{attribute addProperty BoxType "EP2328-1061-0016"}
{attribute addProperty Id "DI_X01_Pin4_InputAT %I*DI_X01_Pin4_Input_E4AEF59E810DI_X01_Pin2_InputAT %I*DI_X01_Pin2_Input_E4AEF59E810DI_X02_Pin4_InputAT %I*DI_X02_Pin4_Input_E4AEF59E810DI_X02_Pin2_InputAT %I*DI_X02_Pin2_Input_E4AEF59E810DO_X03_Pin4_OutputAT %Q*DO_X03_Pin4_Output_7F374EB0810DO_X03_Pin2_OutputAT %Q*DO_X03_Pin2_Output_7F374EB0810DO_X04_Pin4_OutputAT %Q*DO_X04_Pin4_Output_7F374EB0810DO_X04_Pin2_OutputAT %Q*DO_X04_Pin2_Output_7F374EB0810WcStateAT %I*WcState_F855686C1620InfoDataAT %I*InfoData_192954DE1620"}
{attribute addProperty CRC "3768556029"}
{attribute addProperty SizeInBites "96"}
{attribute addProperty SizeInBytes "12"}
TYPE EP2328_6092ACCC :
STRUCT
	{attribute addProperty Name "DI_X01_Pin4_Input"}
	DI_X01_Pin4_Input : DI_X01_Pin4_Input_E4AEF59E;
	{attribute addProperty Name "DI_X01_Pin2_Input"}
	DI_X01_Pin2_Input : DI_X01_Pin2_Input_E4AEF59E;
	{attribute addProperty Name "DI_X02_Pin4_Input"}
	DI_X02_Pin4_Input : DI_X02_Pin4_Input_E4AEF59E;
	{attribute addProperty Name "DI_X02_Pin2_Input"}
	DI_X02_Pin2_Input : DI_X02_Pin2_Input_E4AEF59E;
	{attribute addProperty Name "DO_X03_Pin4_Output"}
	DO_X03_Pin4_Output : DO_X03_Pin4_Output_7F374EB0;
	{attribute addProperty Name "DO_X03_Pin2_Output"}
	DO_X03_Pin2_Output : DO_X03_Pin2_Output_7F374EB0;
	{attribute addProperty Name "DO_X04_Pin4_Output"}
	DO_X04_Pin4_Output : DO_X04_Pin4_Output_7F374EB0;
	{attribute addProperty Name "DO_X04_Pin2_Output"}
	DO_X04_Pin2_Output : DO_X04_Pin2_Output_7F374EB0;
	{attribute addProperty Name "WcState"}
	WcState : WcState_F855686C;
	{attribute addProperty Name "InfoData"}
	InfoData : InfoData_192954DE;
END_STRUCT
END_TYPE

(* stored: Version 1.2.0.0, ProductVersion 3.1.4024.9
   DUT EP2328_6092ACCC: Id {4048953e-6aca-4a97-b35e-d920925ebb58} *)
